FUNCTION_BLOCK AX2_X_TO_BOOL (* Composite FB for convert AX2 to BOOL *)
  (* Standard: 61499-2; Description: Copyright (c) 2024 HR Agrartechnik GmbH This program and the accompanying materials are made available under the terms of the Eclipse Public License 2.0 which is available at https://www.eclipse.org/legal/epl-2.0/ SPDX-License-Identifier: EPL-2.0 *)
  (* Version 1.0, 2024-04-24, Franz Höpfinger, HR Agrartechnik GmbH *)
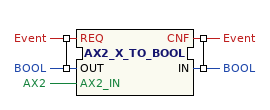
  EVENT_INPUT
    REQ WITH OUT; (* Request to Adapter *)
  END_EVENT
  EVENT_OUTPUT
    CNF WITH IN; (* Confirmation from Adapter *)
  END_EVENT
  VAR_INPUT
    OUT : BOOL;
  END_VAR
  VAR_OUTPUT
    IN : BOOL; (* Input data from Adapter *)
  END_VAR
  SOCKETS
    AX2_IN : AX2; (* Adapter Input *)
  END_SOCKETS
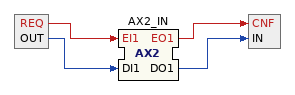
  EVENT_CONNECTIONS
    AX2_IN.EO1 TO CNF;
    REQ TO AX2_IN.EI1;
  END_CONNECTIONS
  DATA_CONNECTIONS
    AX2_IN.DO1 TO IN;
    OUT TO AX2_IN.DI1;
  END_CONNECTIONS
END_FUNCTION_BLOCK
